# EPICS autosave request: ADBruker/brukerApp/Db/BIS_settings.req
$(P)$(R)ReadSFRMTimeout
$(P)$(R)NumDarks
file "ADBASE_settings.req", P=$(P), R=$(R)
file "NDFile_settings.req", P=$(P), R=$(R)
